FUNCTION_BLOCK FB_Generator
VAR_INPUT
END_VAR
VAR_OUTPUT
END_VAR
VAR
	// instance variables
	fbTon1		: TON;	
	tCycletime	: TIME:=T#1S;
	bToggle		: BOOL;

	
	fbTp1		: TP;		
	tPulsetime	: TIME := T#800MS;
END_VAR

PROPERTY Cycletime : TIME
GET
Cycletime := this^.tCycletime;
END_GET
SET
(*Limit Input Value *)
IF Cycletime < T#50MS THEN
	tCycletime := T#50MS;
ELSIF Cycletime > T#5S THEN
	tCycletime := T#5S;
ELSE	
	tCycletime := Cycletime;
END_IF
END_SET
END_PROPERTY

METHOD Flash : BOOL
VAR_INPUT
END_VAR
fbTon1(IN:= NOT fbTon1.Q , PT:=THIS^.tCycletime , Q=> , ET=> );
IF fbTon1.Q THEN
	bToggle:= NOT bToggle;
END_IF
Flash:= bToggle;
END_METHOD

METHOD Pulse : BOOL
VAR_INPUT
	bTriggPuls: BOOL;
END_VAR
fbTp1(IN:=bTriggPuls , PT:=this^.tPulsetime , Q=>Pulse , ET=> );
END_METHOD

PROPERTY Vendor : STRING
GET
Vendor := 'Training';
END_GET
END_PROPERTY

END_FUNCTION_BLOCK

(* stored: Version 1.1.0.1, ProductVersion 3.1.4024.6
   POU FB_Generator: Id {24a43d9d-dd7b-41fd-9822-cc2287b75bcc}, SpecialFunc None
   Property Cycletime: Id {28efd41d-4de4-4a81-af2b-845e86aa7a75}
   Get Get: Id {8f5d3b2b-0044-406b-b6fd-bb47940baec8}
   Set Set: Id {ddf781d1-835a-41ee-afd8-d5276132b0da}
   Method Flash: Id {214c2423-b1b4-4b14-bbd4-9bbe6a541002}
   Method Pulse: Id {8c972a96-a0bf-4042-a12d-e5286d30812f}
   Property Vendor: Id {c6dda2ec-51a2-4469-afe7-640de58907fd}
   Get Get: Id {40d32773-b1f0-47e4-b2b7-a44cbfc9c893} *)
